{attribute addProperty BoxType "EL2521-0000-1017"}
{attribute addProperty Id "StatusAT %I*Status_9C06BD661620Counter_valueAT %I*UINT16217"}
{attribute addProperty CRC "3633927053"}
{attribute addProperty SizeInBites "32"}
{attribute addProperty SizeInBytes "4"}
TYPE ENC_Status_compact_D899538D :
STRUCT
	{attribute addProperty Name "Status"}
	Status AT %I* : Status_9C06BD66;
	{attribute addProperty Name "Counter_value"}
	Counter_value AT %I* : UINT;
END_STRUCT
END_TYPE

(* stored: Version 1.2.0.0, ProductVersion 3.1.4024.9
   DUT ENC_Status_compact_D899538D: Id {431f8be0-effc-40a4-9f85-1deca5ced5a7} *)
